(* PLC project PLC_Kin4DCable, Beckhoff Automation GmbH TwinCAT PLC Control 3.5.13.21 *)
(* stored: creationDateTime 2023-10-16T11:43:55.1345865, modificationDateTime 2023-10-16T11:43:55.1374231 *)

FUNCTION_BLOCK FB_Power
VAR_INPUT
	bEnable			: BOOL := FALSE;
	fOverride		: LREAL := 1.0;
END_VAR
VAR_IN_OUT
	stAxisAcs		: ARRAY[1..4] OF AXIS_REF;
	stAxisMcs		: ARRAY[1..3] OF AXIS_REF;
END_VAR
VAR_OUTPUT
	bAllAxesReady	: BOOL := FALSE;
	bError			: BOOL;
END_VAR
VAR
	fbPowerAcs		: ARRAY [1..4] OF MC_Power;
	fbPowerMcs	 	: ARRAY [1..3] OF MC_Power;
	i				: UINT;
END_VAR

            bAllAxesReady := TRUE;
bError := FALSE;

FOR i:=1 TO 4 DO
	fbPowerAcs[i](Axis:=stAxisAcs[i],
		Enable			:= bEnable,
		Enable_Positive	:= bEnable,
		Enable_Negative	:= bEnable
	);
	
	IF i <= 3 THEN
		fbPowerMcs[i](Axis:=stAxisMcs[i],
			Enable			:= bEnable,
			Enable_Positive	:= bEnable,
			Enable_Negative	:= bEnable
		);
		
		bAllAxesReady := bAllAxesReady AND fbPowerAcs[i].Status AND fbPowerMcs[i].Status; 
		bError := bError OR fbPowerAcs[i].Error OR fbPowerMcs[i].Error;
		
	ELSE
		bAllAxesReady := bAllAxesReady AND fbPowerAcs[i].Status;
		bError := bError OR fbPowerAcs[i].Error;
	END_IF
	 
END_FOR
          
END_FUNCTION_BLOCK

PROGRAM MAIN
VAR
	(* user interaction *)
	bUserStartSequence		: BOOL 	:= FALSE;
	fUserOverride			: LREAL	:= 100.0;
	fUserVelocityToStartPos	: LREAL := 100;
	
	(* *)
	nState					: INT := 0;
	stAxisAcs				: ARRAY[1..4] OF AXIS_REF;
	stAxisMcs				: ARRAY[1..3] OF AXIS_REF;
	
	stKinRefIn    AT %I*	: NCTOPLC_NCICHANNEL_REF;
	stKinRefOut   AT %Q*  	: PLCTONC_NCICHANNEL_REF;
	
	fbPower					: FB_Power;
	fbKinConfigGroup      	: FB_KinConfigGroup;	
	fbKinResetGroup			: FB_KinResetGroup;
	fbKinCalcTrafo			: FB_KinCalcTrafo;
	stKinAxesList          	: ST_KinAxes;
	
		
	fbMoveAbsoluteAx1		: MC_MoveAbsolute;
	fbMoveAbsoluteAx2		: MC_MoveAbsolute;
	fbMoveAbsoluteAx3		: MC_MoveAbsolute;
	fbMoveAbsoluteAx4		: MC_MoveAbsolute;
	
	bBuildKinGroup			: BOOL;
	bPayloadAttached		: BOOL;
END_VAR

            // =========================================
// ToDo: Add Description
// =========================================

ReadAxisStatus();

// Power all axes
fbPower(
	bEnable := TRUE, 
	fOverride := fUserOverride,
	stAxisAcs := stAxisAcs,
	stAxisMcs := stAxisMcs, 
	bAllAxesReady =>,
	bError => );

IF fbPower.bError THEN	
	(* ToDo: add error handling *)
END_IF	

CASE nState OF
0:	// read the IDs from the cyclic axis interface so the axes can mapped later to the kinematic group 
	IF bUserStartSequence AND fbPower.bAllAxesReady THEN
		stKinAxesList.nAxisIdsAcs[1] := stAxisAcs[1].NcToPlc.AxisId;
		stKinAxesList.nAxisIdsAcs[2] := stAxisAcs[2].NcToPlc.AxisId;
		stKinAxesList.nAxisIdsAcs[3] := stAxisAcs[3].NcToPlc.AxisId;
		stKinAxesList.nAxisIdsAcs[4] := stAxisAcs[4].NcToPlc.AxisId;
		
		stKinAxesList.nAxisIdsMcs[1] := stAxisMcs[1].NcToPlc.AxisId;
		stKinAxesList.nAxisIdsMcs[2] := stAxisMcs[2].NcToPlc.AxisId;
		stKinAxesList.nAxisIdsMcs[3] := stAxisMcs[3].NcToPlc.AxisId;
		
		bUserStartSequence := FALSE;
		nState := nState + 10;
	END_IF
	
10:	
	fbMoveAbsoluteAx1(Axis:= stAxisAcs[1], Execute:= TRUE, Position:= 1500, Velocity:= fUserVelocityToStartPos);
	fbMoveAbsoluteAx2(Axis:= stAxisAcs[2], Execute:= TRUE, Position:= 1500, Velocity:= fUserVelocityToStartPos);
	fbMoveAbsoluteAx3(Axis:= stAxisAcs[3], Execute:= TRUE, Position:= 1500, Velocity:= fUserVelocityToStartPos);
	fbMoveAbsoluteAx4(Axis:= stAxisAcs[4], Execute:= TRUE, Position:= 1500, Velocity:= fUserVelocityToStartPos);


	IF fbMoveAbsoluteAx1.Done AND fbMoveAbsoluteAx2.Done AND fbMoveAbsoluteAx3.Done AND fbMoveAbsoluteAx4.Done THEN
		fbMoveAbsoluteAx1( Axis:= stAxisAcs[1], Execute:= FALSE); 
		fbMoveAbsoluteAx2( Axis:= stAxisAcs[2], Execute:= FALSE); 
		fbMoveAbsoluteAx3( Axis:= stAxisAcs[3], Execute:= FALSE); 
		fbMoveAbsoluteAx4( Axis:= stAxisAcs[4], Execute:= FALSE);	
		nState := nState +10;
	ELSIF fbMoveAbsoluteAx1.Error OR fbMoveAbsoluteAx2.Error OR fbMoveAbsoluteAx3.Error OR fbMoveAbsoluteAx4.Error THEN
		(* ToDo: add error handling *)			
		nState := nState +1000;	
	END_IF	
	
20:
	IF bPayloadAttached THEN
		bPayloadAttached := FALSE;
		nState := nState +10;
	END_IF
	
30:	// configure and build kinematic group
	fbKinConfigGroup(
		bExecute       := TRUE,
		bCartesianMode := TRUE,
		stAxesList     := stKinAxesList,
		stKinRefIn     := stKinRefIn ); 
	
	IF fbKinConfigGroup.bDone THEN
		fbKinConfigGroup(bExecute := FALSE, stAxesList := stKinAxesList, stKinRefIn := stKinRefIn);
		nState := nState +10;
	ELSIF fbKinConfigGroup.bError THEN
		(* ToDo: add error handling *)			
		nState := nState +1000;	
	END_IF	
	
1000..9999:
	;//Error				
END_CASE


          

ACTION ReadAxisStatus:
                stAxisAcs[1].ReadStatus();
stAxisAcs[2].ReadStatus();
stAxisAcs[3].ReadStatus();
stAxisMcs[1].ReadStatus();
stAxisMcs[2].ReadStatus();
stAxisMcs[3].ReadStatus();
              
END_ACTION
END_PROGRAM
